// TIA Portal V16 export
// export: Created 2023-06-21T17:06:26.413978Z, ExportSetting WithDefaults, DisplayName Totally Integrated Automation Portal, DisplayVersion V16 Update 4, DisplayName TIA Portal Version Control Interface, DisplayVersion V16 Update 2, DisplayName TIA Portal Openness, DisplayVersion V16 Update 4, DisplayName SINAMICS Startdrive Advanced, DisplayVersion V16, DisplayName SINAMICS Startdrive G130, G150, S120, S150, SINAMICS MV, S210, DisplayVersion V16, DisplayName SINAMICS Startdrive G110M, G120, G120C, G120D, G120P, DisplayVersion V16, DisplayName STEP 7 Professional, DisplayVersion V16 Update 4, DisplayName STEP 7 Safety, DisplayVersion V16, DisplayName Soft Starter ES, DisplayVersion V16, DisplayName WinCC Advanced, DisplayVersion V16 Update 4
FUNCTION_BLOCK "MB_Comm_Setup"   // FB1, LAD
{ S7_Optimized_Access := 'FALSE' }
VERSION : 0.1
// stored: AutoNumber true, IsIECCheckEnabled false, SetENOAutomatically false, UDAEnableTagReadback false
   VAR DB_SPECIFIC
      Input_Registers_3000X_In { ExternalAccessible := 'False'; ExternalVisible := 'False'; ExternalWritable := 'False'} : Struct
         "3000X" { ExternalAccessible := 'False'; ExternalVisible := 'False'; ExternalWritable := 'False'} : Array[0..150] of Word;
      END_STRUCT;
   END_VAR
   VAR
      Input_Registers_In_AT AT Input_Registers_3000X_In : Struct
         "30001" : Array[0..15] of Bool;
         "30001_2" : Array[0..15] of Bool;   // Status of the Adaptor
         "30002" : Array[0..15] of Bool;   // Indoor Unit Connection Status
         "30003" : Array[0..15] of Bool;   // Empty
         "30004" : Array[0..15] of Bool;   // Empty
         "30005" : Array[0..15] of Bool;   // Empty
         "30006" : Array[0..15] of Bool;   // Indoor Unit Communication Status
         "31001" : Array[0..15] of Bool;   // Various
         "31002" : Array[0..15] of Bool;   // 1st word - Indoor unit cooling setpoint upper limit, 2 - word indoor unit cooling setpoint lower limit
         "31003" : Array[0..15] of Bool;   // 1st word - Indoor unit heating setpoint upper limit, 2 - word indoor unit heating setpoint lower limit
         "31004" : Array[0..15] of Bool;   // Various
         "31005" : Array[0..15] of Bool;   // 1st word - Indoor unit cooling setpoint upper limit, 2 - word indoor unit cooling setpoint lower limit
         "31006" : Array[0..15] of Bool;   // 1st word - Indoor unit heating setpoint upper limit, 2 - word indoor unit heating setpoint lower limit
         "31007" : Array[0..15] of Bool;   // Various
         "31008" : Array[0..15] of Bool;   // 1st word - Indoor unit cooling setpoint upper limit, 2 - word indoor unit cooling setpoint lower limit
         "31009" : Array[0..15] of Bool;   // 1st word - Indoor unit heating setpoint upper limit, 2 - word indoor unit heating setpoint lower limit
         "31010" : Array[0..15] of Bool;   // Various
         "31011" : Array[0..15] of Bool;   // 1st word - Indoor unit cooling setpoint upper limit, 2 - word indoor unit cooling setpoint lower limit
         "31012" : Array[0..15] of Bool;   // 1st word - Indoor unit heating setpoint upper limit, 2 - word indoor unit heating setpoint lower limit
         "31013" : Array[0..15] of Bool;   // Various
         "31014" : Array[0..15] of Bool;   // 1st word - Indoor unit cooling setpoint upper limit, 2 - word indoor unit cooling setpoint lower limit
         "31015" : Array[0..15] of Bool;   // 1st word - Indoor unit heating setpoint upper limit, 2 - word indoor unit heating setpoint lower limit
         "31016" : Array[0..15] of Bool;   // Various
         "31017" : Array[0..15] of Bool;   // 1st word - Indoor unit cooling setpoint upper limit, 2 - word indoor unit cooling setpoint lower limit
         "31018" : Array[0..15] of Bool;   // 1st word - Indoor unit heating setpoint upper limit, 2 - word indoor unit heating setpoint lower limit
         "31019" : Array[0..15] of Bool;   // Various
         "31020" : Array[0..15] of Bool;   // 1st word - Indoor unit cooling setpoint upper limit, 2 - word indoor unit cooling setpoint lower limit
         "31021" : Array[0..15] of Bool;   // 1st word - Indoor unit heating setpoint upper limit, 2 - word indoor unit heating setpoint lower limit
         "31022" : Array[0..15] of Bool;   // Various
         "31023" : Array[0..15] of Bool;   // 1st word - Indoor unit cooling setpoint upper limit, 2 - word indoor unit cooling setpoint lower limit
         "31024" : Array[0..15] of Bool;   // 1st word - Indoor unit heating setpoint upper limit, 2 - word indoor unit heating setpoint lower limit
         "31025" : Array[0..15] of Bool;   // Various
         "31026" : Array[0..15] of Bool;   // 1st word - Indoor unit cooling setpoint upper limit, 2 - word indoor unit cooling setpoint lower limit
         "31027" : Array[0..15] of Bool;   // 1st word - Indoor unit heating setpoint upper limit, 2 - word indoor unit heating setpoint lower limit
         "31028" : Array[0..15] of Bool;   // Various
         "31029" : Array[0..15] of Bool;   // 1st word - Indoor unit cooling setpoint upper limit, 2 - word indoor unit cooling setpoint lower limit
         "31030" : Array[0..15] of Bool;   // 1st word - Indoor unit heating setpoint upper limit, 2 - word indoor unit heating setpoint lower limit
         "31031" : Array[0..15] of Bool;   // Various
         "31032" : Array[0..15] of Bool;   // 1st word - Indoor unit cooling setpoint upper limit, 2 - word indoor unit cooling setpoint lower limit
         "31033" : Array[0..15] of Bool;   // 1st word - Indoor unit heating setpoint upper limit, 2 - word indoor unit heating setpoint lower limit
         "31034" : Array[0..15] of Bool;   // Various
         "31035" : Array[0..15] of Bool;   // 1st word - Indoor unit cooling setpoint upper limit, 2 - word indoor unit cooling setpoint lower limit
         "31036" : Array[0..15] of Bool;   // 1st word - Indoor unit heating setpoint upper limit, 2 - word indoor unit heating setpoint lower limit
         "31037" : Array[0..15] of Bool;   // Various
         "31038" : Array[0..15] of Bool;   // 1st word - Indoor unit cooling setpoint upper limit, 2 - word indoor unit cooling setpoint lower limit
         "31039" : Array[0..15] of Bool;   // 1st word - Indoor unit heating setpoint upper limit, 2 - word indoor unit heating setpoint lower limit
         "31040" : Array[0..15] of Bool;   // Various
         "31041" : Array[0..15] of Bool;   // 1st word - Indoor unit cooling setpoint upper limit, 2 - word indoor unit cooling setpoint lower limit
         "31042" : Array[0..15] of Bool;   // 1st word - Indoor unit heating setpoint upper limit, 2 - word indoor unit heating setpoint lower limit
         "31043" : Array[0..15] of Bool;   // Various
         "31044" : Array[0..15] of Bool;   // 1st word - Indoor unit cooling setpoint upper limit, 2 - word indoor unit cooling setpoint lower limit
         "31045" : Array[0..15] of Bool;   // 1st word - Indoor unit heating setpoint upper limit, 2 - word indoor unit heating setpoint lower limit
         "31046" : Array[0..15] of Bool;   // Various
         "31047" : Array[0..15] of Bool;   // 1st word - Indoor unit cooling setpoint upper limit, 2 - word indoor unit cooling setpoint lower limit
         "31048" : Array[0..15] of Bool;   // 1st word - Indoor unit heating setpoint upper limit, 2 - word indoor unit heating setpoint lower limit
         "32001" : Array[0..15] of Bool;   // Important stuff
         "32002" : Array[0..15] of Bool;   // Important stuff_2
         "32003" : Array[0..15] of Bool;   // Setpoint Temperature
         "32004" : Array[0..15] of Bool;   // Important Stuff_3
         "32005" : Array[0..15] of Bool;   // Room Temperature
         "32006" : Array[0..15] of Bool;   // Error
         "32007" : Array[0..15] of Bool;   // Important stuff
         "32008" : Array[0..15] of Bool;   // Important stuff_2
         "32009" : Array[0..15] of Bool;   // Setpoint Temperature
         "32010" : Array[0..15] of Bool;   // Important Stuff_3
         "32011" : Array[0..15] of Bool;   // Room Temperature
         "32012" : Array[0..15] of Bool;   // Error
         "32013" : Array[0..15] of Bool;   // Important stuff
         "32014" : Array[0..15] of Bool;   // Important stuff_2
         "32015" : Array[0..15] of Bool;   // Setpoint Temperature
         "32016" : Array[0..15] of Bool;   // Important Stuff_3
         "32017" : Array[0..15] of Bool;   // Room Temperature
         "32018" : Array[0..15] of Bool;   // Error
         "32019" : Array[0..15] of Bool;   // Important stuff
         "32020" : Array[0..15] of Bool;   // Important stuff_2
         "32021" : Array[0..15] of Bool;   // Setpoint Temperature
         "32022" : Array[0..15] of Bool;   // Important Stuff_3
         "32023" : Array[0..15] of Bool;   // Room Temperature
         "32024" : Array[0..15] of Bool;   // Error
         "32025" : Array[0..15] of Bool;   // Important stuff
         "32026" : Array[0..15] of Bool;   // Important stuff_2
         "32027" : Array[0..15] of Bool;   // Setpoint Temperature
         "32028" : Array[0..15] of Bool;   // Important Stuff_3
         "32029" : Array[0..15] of Bool;   // Room Temperature
         "32030" : Array[0..15] of Bool;   // Error
         "32031" : Array[0..15] of Bool;   // Important stuff
         "32032" : Array[0..15] of Bool;   // Important stuff_2
         "32033" : Array[0..15] of Bool;   // Setpoint Temperature
         "32034" : Array[0..15] of Bool;   // Important Stuff_3
         "32035" : Array[0..15] of Bool;   // Room Temperature
         "32036" : Array[0..15] of Bool;   // Error
         "32037" : Array[0..15] of Bool;   // Important stuff
         "32038" : Array[0..15] of Bool;   // Important stuff_2
         "32039" : Array[0..15] of Bool;   // Setpoint Temperature
         "32040" : Array[0..15] of Bool;   // Important Stuff_3
         "32041" : Array[0..15] of Bool;   // Room Temperature
         "32042" : Array[0..15] of Bool;   // Error
         "32043" : Array[0..15] of Bool;   // Important stuff
         "32044" : Array[0..15] of Bool;   // Important stuff_2
         "32045" : Array[0..15] of Bool;   // Setpoint Temperature
         "32046" : Array[0..15] of Bool;   // Important Stuff_3
         "32047" : Array[0..15] of Bool;   // Room Temperature
         "32048" : Array[0..15] of Bool;   // Error
         "32049" : Array[0..15] of Bool;   // Important stuff
         "32050" : Array[0..15] of Bool;   // Important stuff_2
         "32051" : Array[0..15] of Bool;   // Setpoint Temperature
         "32052" : Array[0..15] of Bool;   // Important Stuff_3
         "32053" : Array[0..15] of Bool;   // Room Temperature
         "32054" : Array[0..15] of Bool;   // Error
         "32055" : Array[0..15] of Bool;   // Important stuff
         "32056" : Array[0..15] of Bool;   // Important stuff_2
         "32057" : Array[0..15] of Bool;   // Setpoint Temperature
         "32058" : Array[0..15] of Bool;   // Important Stuff_3
         "32059" : Array[0..15] of Bool;   // Room Temperature
         "32060" : Array[0..15] of Bool;   // Error
         "32061" : Array[0..15] of Bool;   // Important stuff
         "32062" : Array[0..15] of Bool;   // Important stuff_2
         "32063" : Array[0..15] of Bool;   // Setpoint Temperature
         "32064" : Array[0..15] of Bool;   // Important Stuff_3
         "32065" : Array[0..15] of Bool;   // Room Temperature
         "32066" : Array[0..15] of Bool;   // Error
         "32067" : Array[0..15] of Bool;   // Important stuff
         "32068" : Array[0..15] of Bool;   // Important stuff_2
         "32069" : Array[0..15] of Bool;   // Setpoint Temperature
         "32070" : Array[0..15] of Bool;   // Important Stuff_3
         "32071" : Array[0..15] of Bool;   // Room Temperature
         "32072" : Array[0..15] of Bool;   // Error
         "32073" : Array[0..15] of Bool;   // Important stuff
         "32074" : Array[0..15] of Bool;   // Important stuff_2
         "32075" : Array[0..15] of Bool;   // Setpoint Temperature
         "32076" : Array[0..15] of Bool;   // Important Stuff_3
         "32077" : Array[0..15] of Bool;   // Room Temperature
         "32078" : Array[0..15] of Bool;   // Error
         "32079" : Array[0..15] of Bool;   // Important stuff
         "32080" : Array[0..15] of Bool;   // Important stuff_2
         "32081" : Array[0..15] of Bool;   // Setpoint Temperature
         "32082" : Array[0..15] of Bool;   // Important Stuff_3
         "32083" : Array[0..15] of Bool;   // Room Temperature
         "32084" : Array[0..15] of Bool;   // Error
         "32085" : Array[0..15] of Bool;   // Important stuff
         "32086" : Array[0..15] of Bool;   // Important stuff_2
         "32087" : Array[0..15] of Bool;   // Setpoint Temperature
         "32088" : Array[0..15] of Bool;   // Important Stuff_3
         "32089" : Array[0..15] of Bool;   // Room Temperature
         "32090" : Array[0..15] of Bool;   // Error
         "32091" : Array[0..15] of Bool;   // Important stuff
         "32092" : Array[0..15] of Bool;   // Important stuff_2
         "32093" : Array[0..15] of Bool;   // Setpoint Temperature
         "32094" : Array[0..15] of Bool;   // Important Stuff_3
         "32095" : Array[0..15] of Bool;   // Room Temperature
         "32096" : Array[0..15] of Bool;   // Error
      END_STRUCT;
   END_VAR
   // // Input_Registers_3000X_In."3000X"[0] : 30001
   // // Input_Registers_In_AT."30004"[0] : Fan Mode Capability
   // // Input_Registers_In_AT."30004"[1] : Cooling Mode Capability
   // // Input_Registers_In_AT."30004"[2] : Heating Mode Capability
   // // Input_Registers_In_AT."30004"[3] : Auto Mode Capability
   // // Input_Registers_In_AT."30004"[4] : Dry Mode Capability
   // // Input_Registers_In_AT."30004"[8] : Fan Direction Level Capability
   // // Input_Registers_In_AT."30004"[9] : Fan Direction Level Capability
   // // Input_Registers_In_AT."30004"[10] : Fan Direction Level Capability
   // // Input_Registers_In_AT."30004"[11] : Fan Direction Capability
   // // Input_Registers_In_AT."30004"[12] : Fan Volume Level Capability
   // // Input_Registers_In_AT."30004"[13] : Fan Volume Level Capability
   // // Input_Registers_In_AT."30004"[14] : Fan Volume Level Capability
   // // Input_Registers_In_AT."30004"[15] : Fan Volume Capability
   // // Input_Registers_In_AT."30005"[0] : Fan Mode Capability
   // // Input_Registers_In_AT."30005"[1] : Cooling Mode Capability
   // // Input_Registers_In_AT."30005"[2] : Heating Mode Capability
   // // Input_Registers_In_AT."30005"[3] : Auto Mode Capability
   // // Input_Registers_In_AT."30005"[4] : Dry Mode Capability
   // // Input_Registers_In_AT."30005"[8] : Fan Direction Level Capability
   // // Input_Registers_In_AT."30005"[9] : Fan Direction Level Capability
   // // Input_Registers_In_AT."30005"[10] : Fan Direction Level Capability
   // // Input_Registers_In_AT."30005"[11] : Fan Direction Capability
   // // Input_Registers_In_AT."30005"[12] : Fan Volume Level Capability
   // // Input_Registers_In_AT."30005"[13] : Fan Volume Level Capability
   // // Input_Registers_In_AT."30005"[14] : Fan Volume Level Capability
   // // Input_Registers_In_AT."30005"[15] : Fan Volume Capability
   // // Input_Registers_In_AT."31001"[0] : Fan Mode Capability
   // // Input_Registers_In_AT."31001"[1] : Cooling Mode Capability
   // // Input_Registers_In_AT."31001"[2] : Heating Mode Capability
   // // Input_Registers_In_AT."31001"[3] : Auto Mode Capability
   // // Input_Registers_In_AT."31001"[4] : Dry Mode Capability
   // // Input_Registers_In_AT."31001"[8] : Fan Direction Level Capability
   // // Input_Registers_In_AT."31001"[9] : Fan Direction Level Capability
   // // Input_Registers_In_AT."31001"[10] : Fan Direction Level Capability
   // // Input_Registers_In_AT."31001"[11] : Fan Direction Capability
   // // Input_Registers_In_AT."31001"[12] : Fan Volume Level Capability
   // // Input_Registers_In_AT."31001"[13] : Fan Volume Level Capability
   // // Input_Registers_In_AT."31001"[14] : Fan Volume Level Capability
   // // Input_Registers_In_AT."31001"[15] : Fan Volume Capability
   // // Input_Registers_In_AT."31004"[0] : Fan Mode Capability
   // // Input_Registers_In_AT."31004"[1] : Cooling Mode Capability
   // // Input_Registers_In_AT."31004"[2] : Heating Mode Capability
   // // Input_Registers_In_AT."31004"[3] : Auto Mode Capability
   // // Input_Registers_In_AT."31004"[4] : Dry Mode Capability
   // // Input_Registers_In_AT."31004"[8] : Fan Direction Level Capability
   // // Input_Registers_In_AT."31004"[9] : Fan Direction Level Capability
   // // Input_Registers_In_AT."31004"[10] : Fan Direction Level Capability
   // // Input_Registers_In_AT."31004"[11] : Fan Direction Capability
   // // Input_Registers_In_AT."31004"[12] : Fan Volume Level Capability
   // // Input_Registers_In_AT."31004"[13] : Fan Volume Level Capability
   // // Input_Registers_In_AT."31004"[14] : Fan Volume Level Capability
   // // Input_Registers_In_AT."31004"[15] : Fan Volume Capability
   // // Input_Registers_In_AT."31007"[0] : Fan Mode Capability
   // // Input_Registers_In_AT."31007"[1] : Cooling Mode Capability
   // // Input_Registers_In_AT."31007"[2] : Heating Mode Capability
   // // Input_Registers_In_AT."31007"[3] : Auto Mode Capability
   // // Input_Registers_In_AT."31007"[4] : Dry Mode Capability
   // // Input_Registers_In_AT."31007"[8] : Fan Direction Level Capability
   // // Input_Registers_In_AT."31007"[9] : Fan Direction Level Capability
   // // Input_Registers_In_AT."31007"[10] : Fan Direction Level Capability
   // // Input_Registers_In_AT."31007"[11] : Fan Direction Capability
   // // Input_Registers_In_AT."31007"[12] : Fan Volume Level Capability
   // // Input_Registers_In_AT."31007"[13] : Fan Volume Level Capability
   // // Input_Registers_In_AT."31007"[14] : Fan Volume Level Capability
   // // Input_Registers_In_AT."31007"[15] : Fan Volume Capability
   // // Input_Registers_In_AT."31010"[0] : Fan Mode Capability
   // // Input_Registers_In_AT."31010"[1] : Cooling Mode Capability
   // // Input_Registers_In_AT."31010"[2] : Heating Mode Capability
   // // Input_Registers_In_AT."31010"[3] : Auto Mode Capability
   // // Input_Registers_In_AT."31010"[4] : Dry Mode Capability
   // // Input_Registers_In_AT."31010"[8] : Fan Direction Level Capability
   // // Input_Registers_In_AT."31010"[9] : Fan Direction Level Capability
   // // Input_Registers_In_AT."31010"[10] : Fan Direction Level Capability
   // // Input_Registers_In_AT."31010"[11] : Fan Direction Capability
   // // Input_Registers_In_AT."31010"[12] : Fan Volume Level Capability
   // // Input_Registers_In_AT."31010"[13] : Fan Volume Level Capability
   // // Input_Registers_In_AT."31010"[14] : Fan Volume Level Capability
   // // Input_Registers_In_AT."31010"[15] : Fan Volume Capability
   // // Input_Registers_In_AT."31013"[0] : Fan Mode Capability
   // // Input_Registers_In_AT."31013"[1] : Cooling Mode Capability
   // // Input_Registers_In_AT."31013"[2] : Heating Mode Capability
   // // Input_Registers_In_AT."31013"[3] : Auto Mode Capability
   // // Input_Registers_In_AT."31013"[4] : Dry Mode Capability
   // // Input_Registers_In_AT."31013"[8] : Fan Direction Level Capability
   // // Input_Registers_In_AT."31013"[9] : Fan Direction Level Capability
   // // Input_Registers_In_AT."31013"[10] : Fan Direction Level Capability
   // // Input_Registers_In_AT."31013"[11] : Fan Direction Capability
   // // Input_Registers_In_AT."31013"[12] : Fan Volume Level Capability
   // // Input_Registers_In_AT."31013"[13] : Fan Volume Level Capability
   // // Input_Registers_In_AT."31013"[14] : Fan Volume Level Capability
   // // Input_Registers_In_AT."31013"[15] : Fan Volume Capability
   // // Input_Registers_In_AT."31016"[0] : Fan Mode Capability
   // // Input_Registers_In_AT."31016"[1] : Cooling Mode Capability
   // // Input_Registers_In_AT."31016"[2] : Heating Mode Capability
   // // Input_Registers_In_AT."31016"[3] : Auto Mode Capability
   // // Input_Registers_In_AT."31016"[4] : Dry Mode Capability
   // // Input_Registers_In_AT."31016"[8] : Fan Direction Level Capability
   // // Input_Registers_In_AT."31016"[9] : Fan Direction Level Capability
   // // Input_Registers_In_AT."31016"[10] : Fan Direction Level Capability
   // // Input_Registers_In_AT."31016"[11] : Fan Direction Capability
   // // Input_Registers_In_AT."31016"[12] : Fan Volume Level Capability
   // // Input_Registers_In_AT."31016"[13] : Fan Volume Level Capability
   // // Input_Registers_In_AT."31016"[14] : Fan Volume Level Capability
   // // Input_Registers_In_AT."31016"[15] : Fan Volume Capability
   // // Input_Registers_In_AT."31019"[0] : Fan Mode Capability
   // // Input_Registers_In_AT."31019"[1] : Cooling Mode Capability
   // // Input_Registers_In_AT."31019"[2] : Heating Mode Capability
   // // Input_Registers_In_AT."31019"[3] : Auto Mode Capability
   // // Input_Registers_In_AT."31019"[4] : Dry Mode Capability
   // // Input_Registers_In_AT."31019"[8] : Fan Direction Level Capability
   // // Input_Registers_In_AT."31019"[9] : Fan Direction Level Capability
   // // Input_Registers_In_AT."31019"[10] : Fan Direction Level Capability
   // // Input_Registers_In_AT."31019"[11] : Fan Direction Capability
   // // Input_Registers_In_AT."31019"[12] : Fan Volume Level Capability
   // // Input_Registers_In_AT."31019"[13] : Fan Volume Level Capability
   // // Input_Registers_In_AT."31019"[14] : Fan Volume Level Capability
   // // Input_Registers_In_AT."31019"[15] : Fan Volume Capability
   // // Input_Registers_In_AT."31022"[0] : Fan Mode Capability
   // // Input_Registers_In_AT."31022"[1] : Cooling Mode Capability
   // // Input_Registers_In_AT."31022"[2] : Heating Mode Capability
   // // Input_Registers_In_AT."31022"[3] : Auto Mode Capability
   // // Input_Registers_In_AT."31022"[4] : Dry Mode Capability
   // // Input_Registers_In_AT."31022"[8] : Fan Direction Level Capability
   // // Input_Registers_In_AT."31022"[9] : Fan Direction Level Capability
   // // Input_Registers_In_AT."31022"[10] : Fan Direction Level Capability
   // // Input_Registers_In_AT."31022"[11] : Fan Direction Capability
   // // Input_Registers_In_AT."31022"[12] : Fan Volume Level Capability
   // // Input_Registers_In_AT."31022"[13] : Fan Volume Level Capability
   // // Input_Registers_In_AT."31022"[14] : Fan Volume Level Capability
   // // Input_Registers_In_AT."31022"[15] : Fan Volume Capability
   // // Input_Registers_In_AT."31025"[0] : Fan Mode Capability
   // // Input_Registers_In_AT."31025"[1] : Cooling Mode Capability
   // // Input_Registers_In_AT."31025"[2] : Heating Mode Capability
   // // Input_Registers_In_AT."31025"[3] : Auto Mode Capability
   // // Input_Registers_In_AT."31025"[4] : Dry Mode Capability
   // // Input_Registers_In_AT."31025"[8] : Fan Direction Level Capability
   // // Input_Registers_In_AT."31025"[9] : Fan Direction Level Capability
   // // Input_Registers_In_AT."31025"[10] : Fan Direction Level Capability
   // // Input_Registers_In_AT."31025"[11] : Fan Direction Capability
   // // Input_Registers_In_AT."31025"[12] : Fan Volume Level Capability
   // // Input_Registers_In_AT."31025"[13] : Fan Volume Level Capability
   // // Input_Registers_In_AT."31025"[14] : Fan Volume Level Capability
   // // Input_Registers_In_AT."31025"[15] : Fan Volume Capability
   // // Input_Registers_In_AT."31028"[0] : Fan Mode Capability
   // // Input_Registers_In_AT."31028"[1] : Cooling Mode Capability
   // // Input_Registers_In_AT."31028"[2] : Heating Mode Capability
   // // Input_Registers_In_AT."31028"[3] : Auto Mode Capability
   // // Input_Registers_In_AT."31028"[4] : Dry Mode Capability
   // // Input_Registers_In_AT."31028"[8] : Fan Direction Level Capability
   // // Input_Registers_In_AT."31028"[9] : Fan Direction Level Capability
   // // Input_Registers_In_AT."31028"[10] : Fan Direction Level Capability
   // // Input_Registers_In_AT."31028"[11] : Fan Direction Capability
   // // Input_Registers_In_AT."31028"[12] : Fan Volume Level Capability
   // // Input_Registers_In_AT."31028"[13] : Fan Volume Level Capability
   // // Input_Registers_In_AT."31028"[14] : Fan Volume Level Capability
   // // Input_Registers_In_AT."31028"[15] : Fan Volume Capability
   // // Input_Registers_In_AT."31031"[0] : Fan Mode Capability
   // // Input_Registers_In_AT."31031"[1] : Cooling Mode Capability
   // // Input_Registers_In_AT."31031"[2] : Heating Mode Capability
   // // Input_Registers_In_AT."31031"[3] : Auto Mode Capability
   // // Input_Registers_In_AT."31031"[4] : Dry Mode Capability
   // // Input_Registers_In_AT."31031"[8] : Fan Direction Level Capability
   // // Input_Registers_In_AT."31031"[9] : Fan Direction Level Capability
   // // Input_Registers_In_AT."31031"[10] : Fan Direction Level Capability
   // // Input_Registers_In_AT."31031"[11] : Fan Direction Capability
   // // Input_Registers_In_AT."31031"[12] : Fan Volume Level Capability
   // // Input_Registers_In_AT."31031"[13] : Fan Volume Level Capability
   // // Input_Registers_In_AT."31031"[14] : Fan Volume Level Capability
   // // Input_Registers_In_AT."31031"[15] : Fan Volume Capability
   // // Input_Registers_In_AT."31034"[0] : Fan Mode Capability
   // // Input_Registers_In_AT."31034"[1] : Cooling Mode Capability
   // // Input_Registers_In_AT."31034"[2] : Heating Mode Capability
   // // Input_Registers_In_AT."31034"[3] : Auto Mode Capability
   // // Input_Registers_In_AT."31034"[4] : Dry Mode Capability
   // // Input_Registers_In_AT."31034"[8] : Fan Direction Level Capability
   // // Input_Registers_In_AT."31034"[9] : Fan Direction Level Capability
   // // Input_Registers_In_AT."31034"[10] : Fan Direction Level Capability
   // // Input_Registers_In_AT."31034"[11] : Fan Direction Capability
   // // Input_Registers_In_AT."31034"[12] : Fan Volume Level Capability
   // // Input_Registers_In_AT."31034"[13] : Fan Volume Level Capability
   // // Input_Registers_In_AT."31034"[14] : Fan Volume Level Capability
   // // Input_Registers_In_AT."31034"[15] : Fan Volume Capability
   // // Input_Registers_In_AT."31037"[0] : Fan Mode Capability
   // // Input_Registers_In_AT."31037"[1] : Cooling Mode Capability
   // // Input_Registers_In_AT."31037"[2] : Heating Mode Capability
   // // Input_Registers_In_AT."31037"[3] : Auto Mode Capability
   // // Input_Registers_In_AT."31037"[4] : Dry Mode Capability
   // // Input_Registers_In_AT."31037"[8] : Fan Direction Level Capability
   // // Input_Registers_In_AT."31037"[9] : Fan Direction Level Capability
   // // Input_Registers_In_AT."31037"[10] : Fan Direction Level Capability
   // // Input_Registers_In_AT."31037"[11] : Fan Direction Capability
   // // Input_Registers_In_AT."31037"[12] : Fan Volume Level Capability
   // // Input_Registers_In_AT."31037"[13] : Fan Volume Level Capability
   // // Input_Registers_In_AT."31037"[14] : Fan Volume Level Capability
   // // Input_Registers_In_AT."31037"[15] : Fan Volume Capability
   // // Input_Registers_In_AT."31040"[0] : Fan Mode Capability
   // // Input_Registers_In_AT."31040"[1] : Cooling Mode Capability
   // // Input_Registers_In_AT."31040"[2] : Heating Mode Capability
   // // Input_Registers_In_AT."31040"[3] : Auto Mode Capability
   // // Input_Registers_In_AT."31040"[4] : Dry Mode Capability
   // // Input_Registers_In_AT."31040"[8] : Fan Direction Level Capability
   // // Input_Registers_In_AT."31040"[9] : Fan Direction Level Capability
   // // Input_Registers_In_AT."31040"[10] : Fan Direction Level Capability
   // // Input_Registers_In_AT."31040"[11] : Fan Direction Capability
   // // Input_Registers_In_AT."31040"[12] : Fan Volume Level Capability
   // // Input_Registers_In_AT."31040"[13] : Fan Volume Level Capability
   // // Input_Registers_In_AT."31040"[14] : Fan Volume Level Capability
   // // Input_Registers_In_AT."31040"[15] : Fan Volume Capability
   // // Input_Registers_In_AT."31043"[0] : Fan Mode Capability
   // // Input_Registers_In_AT."31043"[1] : Cooling Mode Capability
   // // Input_Registers_In_AT."31043"[2] : Heating Mode Capability
   // // Input_Registers_In_AT."31043"[3] : Auto Mode Capability
   // // Input_Registers_In_AT."31043"[4] : Dry Mode Capability
   // // Input_Registers_In_AT."31043"[8] : Fan Direction Level Capability
   // // Input_Registers_In_AT."31043"[9] : Fan Direction Level Capability
   // // Input_Registers_In_AT."31043"[10] : Fan Direction Level Capability
   // // Input_Registers_In_AT."31043"[11] : Fan Direction Capability
   // // Input_Registers_In_AT."31043"[12] : Fan Volume Level Capability
   // // Input_Registers_In_AT."31043"[13] : Fan Volume Level Capability
   // // Input_Registers_In_AT."31043"[14] : Fan Volume Level Capability
   // // Input_Registers_In_AT."31043"[15] : Fan Volume Capability
   // // Input_Registers_In_AT."31046"[0] : Fan Mode Capability
   // // Input_Registers_In_AT."31046"[1] : Cooling Mode Capability
   // // Input_Registers_In_AT."31046"[2] : Heating Mode Capability
   // // Input_Registers_In_AT."31046"[3] : Auto Mode Capability
   // // Input_Registers_In_AT."31046"[4] : Dry Mode Capability
   // // Input_Registers_In_AT."31046"[8] : Fan Direction Level Capability
   // // Input_Registers_In_AT."31046"[9] : Fan Direction Level Capability
   // // Input_Registers_In_AT."31046"[10] : Fan Direction Level Capability
   // // Input_Registers_In_AT."31046"[11] : Fan Direction Capability
   // // Input_Registers_In_AT."31046"[12] : Fan Volume Level Capability
   // // Input_Registers_In_AT."31046"[13] : Fan Volume Level Capability
   // // Input_Registers_In_AT."31046"[14] : Fan Volume Level Capability
   // // Input_Registers_In_AT."31046"[15] : Fan Volume Capability
   // // Input_Registers_In_AT."32001"[0] : OnOff Status
   // // Input_Registers_In_AT."32001"[2] : Forced off status
   // // Input_Registers_In_AT."32001"[8] : Fan direction
   // // Input_Registers_In_AT."32001"[9] : Fan direction
   // // Input_Registers_In_AT."32001"[10] : Fan direction
   // // Input_Registers_In_AT."32001"[12] : Fan volume
   // // Input_Registers_In_AT."32001"[13] : Fan volume
   // // Input_Registers_In_AT."32001"[14] : Fan volume
   // // Input_Registers_In_AT."32002"[0] : Operation mode
   // // Input_Registers_In_AT."32002"[1] : Operation mode
   // // Input_Registers_In_AT."32002"[2] : Operation mode
   // // Input_Registers_In_AT."32002"[3] : Operation mode
   // // Input_Registers_In_AT."32002"[4] : Filter sign status
   // // Input_Registers_In_AT."32002"[5] : Filter sign status
   // // Input_Registers_In_AT."32002"[6] : Filter sign status
   // // Input_Registers_In_AT."32002"[7] : Filter sign status
   // // Input_Registers_In_AT."32002"[8] : Operation status
   // // Input_Registers_In_AT."32002"[9] : Operation status
   // // Input_Registers_In_AT."32002"[10] : Operation status
   // // Input_Registers_In_AT."32002"[11] : Operation status
   // // Input_Registers_In_AT."32002"[14] : Cool/Heat Master
   // // Input_Registers_In_AT."32002"[15] : Cool/Heat Master
   // // Input_Registers_In_AT."32003"[15] : Signed Bit
   // // Input_Registers_In_AT."32004"[0] : Error code mapping value1
   // // Input_Registers_In_AT."32004"[1] : Error code mapping value1
   // // Input_Registers_In_AT."32004"[2] : Error code mapping value1
   // // Input_Registers_In_AT."32004"[3] : Error code mapping value1
   // // Input_Registers_In_AT."32004"[4] : Error code mapping value2
   // // Input_Registers_In_AT."32004"[5] : Error code mapping value2
   // // Input_Registers_In_AT."32004"[6] : Error code mapping value2
   // // Input_Registers_In_AT."32004"[7] : Error code mapping value2
   // // Input_Registers_In_AT."32004"[8] : Malfunction
   // // Input_Registers_In_AT."32004"[9] : Warning
   // // Input_Registers_In_AT."32004"[10] : Operation status
   // // Input_Registers_In_AT."32005"[15] : Signed Bit
   // // Input_Registers_In_AT."32006"[8] : Indoor unit temperature sensor error
   // // Input_Registers_In_AT."32006"[15] : Indoor unit temperature sensor data received
   // // Input_Registers_In_AT."32007"[0] : OnOff Status
   // // Input_Registers_In_AT."32007"[2] : Forced off status
   // // Input_Registers_In_AT."32007"[8] : Fan direction
   // // Input_Registers_In_AT."32007"[9] : Fan direction
   // // Input_Registers_In_AT."32007"[10] : Fan direction
   // // Input_Registers_In_AT."32007"[12] : Fan volume
   // // Input_Registers_In_AT."32007"[13] : Fan volume
   // // Input_Registers_In_AT."32007"[14] : Fan volume
   // // Input_Registers_In_AT."32008"[0] : Operation mode
   // // Input_Registers_In_AT."32008"[1] : Operation mode
   // // Input_Registers_In_AT."32008"[2] : Operation mode
   // // Input_Registers_In_AT."32008"[3] : Operation mode
   // // Input_Registers_In_AT."32008"[4] : Filter sign status
   // // Input_Registers_In_AT."32008"[5] : Filter sign status
   // // Input_Registers_In_AT."32008"[6] : Filter sign status
   // // Input_Registers_In_AT."32008"[7] : Filter sign status
   // // Input_Registers_In_AT."32008"[8] : Operation status
   // // Input_Registers_In_AT."32008"[9] : Operation status
   // // Input_Registers_In_AT."32008"[10] : Operation status
   // // Input_Registers_In_AT."32008"[11] : Operation status
   // // Input_Registers_In_AT."32008"[14] : Cool/Heat Master
   // // Input_Registers_In_AT."32008"[15] : Cool/Heat Master
   // // Input_Registers_In_AT."32009"[15] : Signed Bit
   // // Input_Registers_In_AT."32010"[0] : Error code mapping value1
   // // Input_Registers_In_AT."32010"[1] : Error code mapping value1
   // // Input_Registers_In_AT."32010"[2] : Error code mapping value1
   // // Input_Registers_In_AT."32010"[3] : Error code mapping value1
   // // Input_Registers_In_AT."32010"[4] : Error code mapping value2
   // // Input_Registers_In_AT."32010"[5] : Error code mapping value2
   // // Input_Registers_In_AT."32010"[6] : Error code mapping value2
   // // Input_Registers_In_AT."32010"[7] : Error code mapping value2
   // // Input_Registers_In_AT."32010"[8] : Malfunction
   // // Input_Registers_In_AT."32010"[9] : Warning
   // // Input_Registers_In_AT."32010"[10] : Operation status
   // // Input_Registers_In_AT."32011"[15] : Signed Bit
   // // Input_Registers_In_AT."32012"[8] : Indoor unit temperature sensor error
   // // Input_Registers_In_AT."32012"[15] : Indoor unit temperature sensor data received
   // // Input_Registers_In_AT."32013"[0] : OnOff Status
   // // Input_Registers_In_AT."32013"[2] : Forced off status
   // // Input_Registers_In_AT."32013"[8] : Fan direction
   // // Input_Registers_In_AT."32013"[9] : Fan direction
   // // Input_Registers_In_AT."32013"[10] : Fan direction
   // // Input_Registers_In_AT."32013"[12] : Fan volume
   // // Input_Registers_In_AT."32013"[13] : Fan volume
   // // Input_Registers_In_AT."32013"[14] : Fan volume
   // // Input_Registers_In_AT."32014"[0] : Operation mode
   // // Input_Registers_In_AT."32014"[1] : Operation mode
   // // Input_Registers_In_AT."32014"[2] : Operation mode
   // // Input_Registers_In_AT."32014"[3] : Operation mode
   // // Input_Registers_In_AT."32014"[4] : Filter sign status
   // // Input_Registers_In_AT."32014"[5] : Filter sign status
   // // Input_Registers_In_AT."32014"[6] : Filter sign status
   // // Input_Registers_In_AT."32014"[7] : Filter sign status
   // // Input_Registers_In_AT."32014"[8] : Operation status
   // // Input_Registers_In_AT."32014"[9] : Operation status
   // // Input_Registers_In_AT."32014"[10] : Operation status
   // // Input_Registers_In_AT."32014"[11] : Operation status
   // // Input_Registers_In_AT."32014"[14] : Cool/Heat Master
   // // Input_Registers_In_AT."32014"[15] : Cool/Heat Master
   // // Input_Registers_In_AT."32015"[15] : Signed Bit
   // // Input_Registers_In_AT."32016"[0] : Error code mapping value1
   // // Input_Registers_In_AT."32016"[1] : Error code mapping value1
   // // Input_Registers_In_AT."32016"[2] : Error code mapping value1
   // // Input_Registers_In_AT."32016"[3] : Error code mapping value1
   // // Input_Registers_In_AT."32016"[4] : Error code mapping value2
   // // Input_Registers_In_AT."32016"[5] : Error code mapping value2
   // // Input_Registers_In_AT."32016"[6] : Error code mapping value2
   // // Input_Registers_In_AT."32016"[7] : Error code mapping value2
   // // Input_Registers_In_AT."32016"[8] : Malfunction
   // // Input_Registers_In_AT."32016"[9] : Warning
   // // Input_Registers_In_AT."32016"[10] : Operation status
   // // Input_Registers_In_AT."32017"[15] : Signed Bit
   // // Input_Registers_In_AT."32018"[8] : Indoor unit temperature sensor error
   // // Input_Registers_In_AT."32018"[15] : Indoor unit temperature sensor data received
   // // Input_Registers_In_AT."32019"[0] : OnOff Status
   // // Input_Registers_In_AT."32019"[2] : Forced off status
   // // Input_Registers_In_AT."32019"[8] : Fan direction
   // // Input_Registers_In_AT."32019"[9] : Fan direction
   // // Input_Registers_In_AT."32019"[10] : Fan direction
   // // Input_Registers_In_AT."32019"[12] : Fan volume
   // // Input_Registers_In_AT."32019"[13] : Fan volume
   // // Input_Registers_In_AT."32019"[14] : Fan volume
   // // Input_Registers_In_AT."32020"[0] : Operation mode
   // // Input_Registers_In_AT."32020"[1] : Operation mode
   // // Input_Registers_In_AT."32020"[2] : Operation mode
   // // Input_Registers_In_AT."32020"[3] : Operation mode
   // // Input_Registers_In_AT."32020"[4] : Filter sign status
   // // Input_Registers_In_AT."32020"[5] : Filter sign status
   // // Input_Registers_In_AT."32020"[6] : Filter sign status
   // // Input_Registers_In_AT."32020"[7] : Filter sign status
   // // Input_Registers_In_AT."32020"[8] : Operation status
   // // Input_Registers_In_AT."32020"[9] : Operation status
   // // Input_Registers_In_AT."32020"[10] : Operation status
   // // Input_Registers_In_AT."32020"[11] : Operation status
   // // Input_Registers_In_AT."32020"[14] : Cool/Heat Master
   // // Input_Registers_In_AT."32020"[15] : Cool/Heat Master
   // // Input_Registers_In_AT."32021"[15] : Signed Bit
   // // Input_Registers_In_AT."32022"[0] : Error code mapping value1
   // // Input_Registers_In_AT."32022"[1] : Error code mapping value1
   // // Input_Registers_In_AT."32022"[2] : Error code mapping value1
   // // Input_Registers_In_AT."32022"[3] : Error code mapping value1
   // // Input_Registers_In_AT."32022"[4] : Error code mapping value2
   // // Input_Registers_In_AT."32022"[5] : Error code mapping value2
   // // Input_Registers_In_AT."32022"[6] : Error code mapping value2
   // // Input_Registers_In_AT."32022"[7] : Error code mapping value2
   // // Input_Registers_In_AT."32022"[8] : Malfunction
   // // Input_Registers_In_AT."32022"[9] : Warning
   // // Input_Registers_In_AT."32022"[10] : Operation status
   // // Input_Registers_In_AT."32023"[15] : Signed Bit
   // // Input_Registers_In_AT."32024"[8] : Indoor unit temperature sensor error
   // // Input_Registers_In_AT."32024"[15] : Indoor unit temperature sensor data received
   // // Input_Registers_In_AT."32025"[0] : OnOff Status
   // // Input_Registers_In_AT."32025"[2] : Forced off status
   // // Input_Registers_In_AT."32025"[8] : Fan direction
   // // Input_Registers_In_AT."32025"[9] : Fan direction
   // // Input_Registers_In_AT."32025"[10] : Fan direction
   // // Input_Registers_In_AT."32025"[12] : Fan volume
   // // Input_Registers_In_AT."32025"[13] : Fan volume
   // // Input_Registers_In_AT."32025"[14] : Fan volume
   // // Input_Registers_In_AT."32026"[0] : Operation mode
   // // Input_Registers_In_AT."32026"[1] : Operation mode
   // // Input_Registers_In_AT."32026"[2] : Operation mode
   // // Input_Registers_In_AT."32026"[3] : Operation mode
   // // Input_Registers_In_AT."32026"[4] : Filter sign status
   // // Input_Registers_In_AT."32026"[5] : Filter sign status
   // // Input_Registers_In_AT."32026"[6] : Filter sign status
   // // Input_Registers_In_AT."32026"[7] : Filter sign status
   // // Input_Registers_In_AT."32026"[8] : Operation status
   // // Input_Registers_In_AT."32026"[9] : Operation status
   // // Input_Registers_In_AT."32026"[10] : Operation status
   // // Input_Registers_In_AT."32026"[11] : Operation status
   // // Input_Registers_In_AT."32026"[14] : Cool/Heat Master
   // // Input_Registers_In_AT."32026"[15] : Cool/Heat Master
   // // Input_Registers_In_AT."32027"[15] : Signed Bit
   // // Input_Registers_In_AT."32028"[0] : Error code mapping value1
   // // Input_Registers_In_AT."32028"[1] : Error code mapping value1
   // // Input_Registers_In_AT."32028"[2] : Error code mapping value1
   // // Input_Registers_In_AT."32028"[3] : Error code mapping value1
   // // Input_Registers_In_AT."32028"[4] : Error code mapping value2
   // // Input_Registers_In_AT."32028"[5] : Error code mapping value2
   // // Input_Registers_In_AT."32028"[6] : Error code mapping value2
   // // Input_Registers_In_AT."32028"[7] : Error code mapping value2
   // // Input_Registers_In_AT."32028"[8] : Malfunction
   // // Input_Registers_In_AT."32028"[9] : Warning
   // // Input_Registers_In_AT."32028"[10] : Operation status
   // // Input_Registers_In_AT."32029"[15] : Signed Bit
   // // Input_Registers_In_AT."32030"[8] : Indoor unit temperature sensor error
   // // Input_Registers_In_AT."32030"[15] : Indoor unit temperature sensor data received
   // // Input_Registers_In_AT."32031"[0] : OnOff Status
   // // Input_Registers_In_AT."32031"[2] : Forced off status
   // // Input_Registers_In_AT."32031"[8] : Fan direction
   // // Input_Registers_In_AT."32031"[9] : Fan direction
   // // Input_Registers_In_AT."32031"[10] : Fan direction
   // // Input_Registers_In_AT."32031"[12] : Fan volume
   // // Input_Registers_In_AT."32031"[13] : Fan volume
   // // Input_Registers_In_AT."32031"[14] : Fan volume
   // // Input_Registers_In_AT."32032"[0] : Operation mode
   // // Input_Registers_In_AT."32032"[1] : Operation mode
   // // Input_Registers_In_AT."32032"[2] : Operation mode
   // // Input_Registers_In_AT."32032"[3] : Operation mode
   // // Input_Registers_In_AT."32032"[4] : Filter sign status
   // // Input_Registers_In_AT."32032"[5] : Filter sign status
   // // Input_Registers_In_AT."32032"[6] : Filter sign status
   // // Input_Registers_In_AT."32032"[7] : Filter sign status
   // // Input_Registers_In_AT."32032"[8] : Operation status
   // // Input_Registers_In_AT."32032"[9] : Operation status
   // // Input_Registers_In_AT."32032"[10] : Operation status
   // // Input_Registers_In_AT."32032"[11] : Operation status
   // // Input_Registers_In_AT."32032"[14] : Cool/Heat Master
   // // Input_Registers_In_AT."32032"[15] : Cool/Heat Master
   // // Input_Registers_In_AT."32033"[15] : Signed Bit
   // // Input_Registers_In_AT."32034"[0] : Error code mapping value1
   // // Input_Registers_In_AT."32034"[1] : Error code mapping value1
   // // Input_Registers_In_AT."32034"[2] : Error code mapping value1
   // // Input_Registers_In_AT."32034"[3] : Error code mapping value1
   // // Input_Registers_In_AT."32034"[4] : Error code mapping value2
   // // Input_Registers_In_AT."32034"[5] : Error code mapping value2
   // // Input_Registers_In_AT."32034"[6] : Error code mapping value2
   // // Input_Registers_In_AT."32034"[7] : Error code mapping value2
   // // Input_Registers_In_AT."32034"[8] : Malfunction
   // // Input_Registers_In_AT."32034"[9] : Warning
   // // Input_Registers_In_AT."32034"[10] : Operation status
   // // Input_Registers_In_AT."32035"[15] : Signed Bit
   // // Input_Registers_In_AT."32036"[8] : Indoor unit temperature sensor error
   // // Input_Registers_In_AT."32036"[15] : Indoor unit temperature sensor data received
   // // Input_Registers_In_AT."32037"[0] : OnOff Status
   // // Input_Registers_In_AT."32037"[2] : Forced off status
   // // Input_Registers_In_AT."32037"[8] : Fan direction
   // // Input_Registers_In_AT."32037"[9] : Fan direction
   // // Input_Registers_In_AT."32037"[10] : Fan direction
   // // Input_Registers_In_AT."32037"[12] : Fan volume
   // // Input_Registers_In_AT."32037"[13] : Fan volume
   // // Input_Registers_In_AT."32037"[14] : Fan volume
   // // Input_Registers_In_AT."32038"[0] : Operation mode
   // // Input_Registers_In_AT."32038"[1] : Operation mode
   // // Input_Registers_In_AT."32038"[2] : Operation mode
   // // Input_Registers_In_AT."32038"[3] : Operation mode
   // // Input_Registers_In_AT."32038"[4] : Filter sign status
   // // Input_Registers_In_AT."32038"[5] : Filter sign status
   // // Input_Registers_In_AT."32038"[6] : Filter sign status
   // // Input_Registers_In_AT."32038"[7] : Filter sign status
   // // Input_Registers_In_AT."32038"[8] : Operation status
   // // Input_Registers_In_AT."32038"[9] : Operation status
   // // Input_Registers_In_AT."32038"[10] : Operation status
   // // Input_Registers_In_AT."32038"[11] : Operation status
   // // Input_Registers_In_AT."32038"[14] : Cool/Heat Master
   // // Input_Registers_In_AT."32038"[15] : Cool/Heat Master
   // // Input_Registers_In_AT."32039"[15] : Signed Bit
   // // Input_Registers_In_AT."32040"[0] : Error code mapping value1
   // // Input_Registers_In_AT."32040"[1] : Error code mapping value1
   // // Input_Registers_In_AT."32040"[2] : Error code mapping value1
   // // Input_Registers_In_AT."32040"[3] : Error code mapping value1
   // // Input_Registers_In_AT."32040"[4] : Error code mapping value2
   // // Input_Registers_In_AT."32040"[5] : Error code mapping value2
   // // Input_Registers_In_AT."32040"[6] : Error code mapping value2
   // // Input_Registers_In_AT."32040"[7] : Error code mapping value2
   // // Input_Registers_In_AT."32040"[8] : Malfunction
   // // Input_Registers_In_AT."32040"[9] : Warning
   // // Input_Registers_In_AT."32040"[10] : Operation status
   // // Input_Registers_In_AT."32041"[15] : Signed Bit
   // // Input_Registers_In_AT."32042"[8] : Indoor unit temperature sensor error
   // // Input_Registers_In_AT."32042"[15] : Indoor unit temperature sensor data received
   // // Input_Registers_In_AT."32043"[0] : OnOff Status
   // // Input_Registers_In_AT."32043"[2] : Forced off status
   // // Input_Registers_In_AT."32043"[8] : Fan direction
   // // Input_Registers_In_AT."32043"[9] : Fan direction
   // // Input_Registers_In_AT."32043"[10] : Fan direction
   // // Input_Registers_In_AT."32043"[12] : Fan volume
   // // Input_Registers_In_AT."32043"[13] : Fan volume
   // // Input_Registers_In_AT."32043"[14] : Fan volume
   // // Input_Registers_In_AT."32044"[0] : Operation mode
   // // Input_Registers_In_AT."32044"[1] : Operation mode
   // // Input_Registers_In_AT."32044"[2] : Operation mode
   // // Input_Registers_In_AT."32044"[3] : Operation mode
   // // Input_Registers_In_AT."32044"[4] : Filter sign status
   // // Input_Registers_In_AT."32044"[5] : Filter sign status
   // // Input_Registers_In_AT."32044"[6] : Filter sign status
   // // Input_Registers_In_AT."32044"[7] : Filter sign status
   // // Input_Registers_In_AT."32044"[8] : Operation status
   // // Input_Registers_In_AT."32044"[9] : Operation status
   // // Input_Registers_In_AT."32044"[10] : Operation status
   // // Input_Registers_In_AT."32044"[11] : Operation status
   // // Input_Registers_In_AT."32044"[14] : Cool/Heat Master
   // // Input_Registers_In_AT."32044"[15] : Cool/Heat Master
   // // Input_Registers_In_AT."32045"[15] : Signed Bit
   // // Input_Registers_In_AT."32046"[0] : Error code mapping value1
   // // Input_Registers_In_AT."32046"[1] : Error code mapping value1
   // // Input_Registers_In_AT."32046"[2] : Error code mapping value1
   // // Input_Registers_In_AT."32046"[3] : Error code mapping value1
   // // Input_Registers_In_AT."32046"[4] : Error code mapping value2
   // // Input_Registers_In_AT."32046"[5] : Error code mapping value2
   // // Input_Registers_In_AT."32046"[6] : Error code mapping value2
   // // Input_Registers_In_AT."32046"[7] : Error code mapping value2
   // // Input_Registers_In_AT."32046"[8] : Malfunction
   // // Input_Registers_In_AT."32046"[9] : Warning
   // // Input_Registers_In_AT."32046"[10] : Operation status
   // // Input_Registers_In_AT."32047"[15] : Signed Bit
   // // Input_Registers_In_AT."32048"[8] : Indoor unit temperature sensor error
   // // Input_Registers_In_AT."32048"[15] : Indoor unit temperature sensor data received
   // // Input_Registers_In_AT."32049"[0] : OnOff Status
   // // Input_Registers_In_AT."32049"[2] : Forced off status
   // // Input_Registers_In_AT."32049"[8] : Fan direction
   // // Input_Registers_In_AT."32049"[9] : Fan direction
   // // Input_Registers_In_AT."32049"[10] : Fan direction
   // // Input_Registers_In_AT."32049"[12] : Fan volume
   // // Input_Registers_In_AT."32049"[13] : Fan volume
   // // Input_Registers_In_AT."32049"[14] : Fan volume
   // // Input_Registers_In_AT."32050"[0] : Operation mode
   // // Input_Registers_In_AT."32050"[1] : Operation mode
   // // Input_Registers_In_AT."32050"[2] : Operation mode
   // // Input_Registers_In_AT."32050"[3] : Operation mode
   // // Input_Registers_In_AT."32050"[4] : Filter sign status
   // // Input_Registers_In_AT."32050"[5] : Filter sign status
   // // Input_Registers_In_AT."32050"[6] : Filter sign status
   // // Input_Registers_In_AT."32050"[7] : Filter sign status
   // // Input_Registers_In_AT."32050"[8] : Operation status
   // // Input_Registers_In_AT."32050"[9] : Operation status
   // // Input_Registers_In_AT."32050"[10] : Operation status
   // // Input_Registers_In_AT."32050"[11] : Operation status
   // // Input_Registers_In_AT."32050"[14] : Cool/Heat Master
   // // Input_Registers_In_AT."32050"[15] : Cool/Heat Master
   // // Input_Registers_In_AT."32051"[15] : Signed Bit
   // // Input_Registers_In_AT."32052"[0] : Error code mapping value1
   // // Input_Registers_In_AT."32052"[1] : Error code mapping value1
   // // Input_Registers_In_AT."32052"[2] : Error code mapping value1
   // // Input_Registers_In_AT."32052"[3] : Error code mapping value1
   // // Input_Registers_In_AT."32052"[4] : Error code mapping value2
   // // Input_Registers_In_AT."32052"[5] : Error code mapping value2
   // // Input_Registers_In_AT."32052"[6] : Error code mapping value2
   // // Input_Registers_In_AT."32052"[7] : Error code mapping value2
   // // Input_Registers_In_AT."32052"[8] : Malfunction
   // // Input_Registers_In_AT."32052"[9] : Warning
   // // Input_Registers_In_AT."32052"[10] : Operation status
   // // Input_Registers_In_AT."32053"[15] : Signed Bit
   // // Input_Registers_In_AT."32054"[8] : Indoor unit temperature sensor error
   // // Input_Registers_In_AT."32054"[15] : Indoor unit temperature sensor data received
   // // Input_Registers_In_AT."32055"[0] : OnOff Status
   // // Input_Registers_In_AT."32055"[2] : Forced off status
   // // Input_Registers_In_AT."32055"[8] : Fan direction
   // // Input_Registers_In_AT."32055"[9] : Fan direction
   // // Input_Registers_In_AT."32055"[10] : Fan direction
   // // Input_Registers_In_AT."32055"[12] : Fan volume
   // // Input_Registers_In_AT."32055"[13] : Fan volume
   // // Input_Registers_In_AT."32055"[14] : Fan volume
   // // Input_Registers_In_AT."32056"[0] : Operation mode
   // // Input_Registers_In_AT."32056"[1] : Operation mode
   // // Input_Registers_In_AT."32056"[2] : Operation mode
   // // Input_Registers_In_AT."32056"[3] : Operation mode
   // // Input_Registers_In_AT."32056"[4] : Filter sign status
   // // Input_Registers_In_AT."32056"[5] : Filter sign status
   // // Input_Registers_In_AT."32056"[6] : Filter sign status
   // // Input_Registers_In_AT."32056"[7] : Filter sign status
   // // Input_Registers_In_AT."32056"[8] : Operation status
   // // Input_Registers_In_AT."32056"[9] : Operation status
   // // Input_Registers_In_AT."32056"[10] : Operation status
   // // Input_Registers_In_AT."32056"[11] : Operation status
   // // Input_Registers_In_AT."32056"[14] : Cool/Heat Master
   // // Input_Registers_In_AT."32056"[15] : Cool/Heat Master
   // // Input_Registers_In_AT."32057"[15] : Signed Bit
   // // Input_Registers_In_AT."32058"[0] : Error code mapping value1
   // // Input_Registers_In_AT."32058"[1] : Error code mapping value1
   // // Input_Registers_In_AT."32058"[2] : Error code mapping value1
   // // Input_Registers_In_AT."32058"[3] : Error code mapping value1
   // // Input_Registers_In_AT."32058"[4] : Error code mapping value2
   // // Input_Registers_In_AT."32058"[5] : Error code mapping value2
   // // Input_Registers_In_AT."32058"[6] : Error code mapping value2
   // // Input_Registers_In_AT."32058"[7] : Error code mapping value2
   // // Input_Registers_In_AT."32058"[8] : Malfunction
   // // Input_Registers_In_AT."32058"[9] : Warning
   // // Input_Registers_In_AT."32058"[10] : Operation status
   // // Input_Registers_In_AT."32059"[15] : Signed Bit
   // // Input_Registers_In_AT."32060"[8] : Indoor unit temperature sensor error
   // // Input_Registers_In_AT."32060"[15] : Indoor unit temperature sensor data received
   // // Input_Registers_In_AT."32061"[0] : OnOff Status
   // // Input_Registers_In_AT."32061"[2] : Forced off status
   // // Input_Registers_In_AT."32061"[8] : Fan direction
   // // Input_Registers_In_AT."32061"[9] : Fan direction
   // // Input_Registers_In_AT."32061"[10] : Fan direction
   // // Input_Registers_In_AT."32061"[12] : Fan volume
   // // Input_Registers_In_AT."32061"[13] : Fan volume
   // // Input_Registers_In_AT."32061"[14] : Fan volume
   // // Input_Registers_In_AT."32062"[0] : Operation mode
   // // Input_Registers_In_AT."32062"[1] : Operation mode
   // // Input_Registers_In_AT."32062"[2] : Operation mode
   // // Input_Registers_In_AT."32062"[3] : Operation mode
   // // Input_Registers_In_AT."32062"[4] : Filter sign status
   // // Input_Registers_In_AT."32062"[5] : Filter sign status
   // // Input_Registers_In_AT."32062"[6] : Filter sign status
   // // Input_Registers_In_AT."32062"[7] : Filter sign status
   // // Input_Registers_In_AT."32062"[8] : Operation status
   // // Input_Registers_In_AT."32062"[9] : Operation status
   // // Input_Registers_In_AT."32062"[10] : Operation status
   // // Input_Registers_In_AT."32062"[11] : Operation status
   // // Input_Registers_In_AT."32062"[14] : Cool/Heat Master
   // // Input_Registers_In_AT."32062"[15] : Cool/Heat Master
   // // Input_Registers_In_AT."32063"[15] : Signed Bit
   // // Input_Registers_In_AT."32064"[0] : Error code mapping value1
   // // Input_Registers_In_AT."32064"[1] : Error code mapping value1
   // // Input_Registers_In_AT."32064"[2] : Error code mapping value1
   // // Input_Registers_In_AT."32064"[3] : Error code mapping value1
   // // Input_Registers_In_AT."32064"[4] : Error code mapping value2
   // // Input_Registers_In_AT."32064"[5] : Error code mapping value2
   // // Input_Registers_In_AT."32064"[6] : Error code mapping value2
   // // Input_Registers_In_AT."32064"[7] : Error code mapping value2
   // // Input_Registers_In_AT."32064"[8] : Malfunction
   // // Input_Registers_In_AT."32064"[9] : Warning
   // // Input_Registers_In_AT."32064"[10] : Operation status
   // // Input_Registers_In_AT."32065"[15] : Signed Bit
   // // Input_Registers_In_AT."32066"[8] : Indoor unit temperature sensor error
   // // Input_Registers_In_AT."32066"[15] : Indoor unit temperature sensor data received
   // // Input_Registers_In_AT."32067"[0] : OnOff Status
   // // Input_Registers_In_AT."32067"[2] : Forced off status
   // // Input_Registers_In_AT."32067"[8] : Fan direction
   // // Input_Registers_In_AT."32067"[9] : Fan direction
   // // Input_Registers_In_AT."32067"[10] : Fan direction
   // // Input_Registers_In_AT."32067"[12] : Fan volume
   // // Input_Registers_In_AT."32067"[13] : Fan volume
   // // Input_Registers_In_AT."32067"[14] : Fan volume
   // // Input_Registers_In_AT."32068"[0] : Operation mode
   // // Input_Registers_In_AT."32068"[1] : Operation mode
   // // Input_Registers_In_AT."32068"[2] : Operation mode
   // // Input_Registers_In_AT."32068"[3] : Operation mode
   // // Input_Registers_In_AT."32068"[4] : Filter sign status
   // // Input_Registers_In_AT."32068"[5] : Filter sign status
   // // Input_Registers_In_AT."32068"[6] : Filter sign status
   // // Input_Registers_In_AT."32068"[7] : Filter sign status
   // // Input_Registers_In_AT."32068"[8] : Operation status
   // // Input_Registers_In_AT."32068"[9] : Operation status
   // // Input_Registers_In_AT."32068"[10] : Operation status
   // // Input_Registers_In_AT."32068"[11] : Operation status
   // // Input_Registers_In_AT."32068"[14] : Cool/Heat Master
   // // Input_Registers_In_AT."32068"[15] : Cool/Heat Master
   // // Input_Registers_In_AT."32069"[15] : Signed Bit
   // // Input_Registers_In_AT."32070"[0] : Error code mapping value1
   // // Input_Registers_In_AT."32070"[1] : Error code mapping value1
   // // Input_Registers_In_AT."32070"[2] : Error code mapping value1
   // // Input_Registers_In_AT."32070"[3] : Error code mapping value1
   // // Input_Registers_In_AT."32070"[4] : Error code mapping value2
   // // Input_Registers_In_AT."32070"[5] : Error code mapping value2
   // // Input_Registers_In_AT."32070"[6] : Error code mapping value2
   // // Input_Registers_In_AT."32070"[7] : Error code mapping value2
   // // Input_Registers_In_AT."32070"[8] : Malfunction
   // // Input_Registers_In_AT."32070"[9] : Warning
   // // Input_Registers_In_AT."32070"[10] : Operation status
   // // Input_Registers_In_AT."32071"[15] : Signed Bit
   // // Input_Registers_In_AT."32072"[8] : Indoor unit temperature sensor error
   // // Input_Registers_In_AT."32072"[15] : Indoor unit temperature sensor data received
   // // Input_Registers_In_AT."32073"[0] : OnOff Status
   // // Input_Registers_In_AT."32073"[2] : Forced off status
   // // Input_Registers_In_AT."32073"[8] : Fan direction
   // // Input_Registers_In_AT."32073"[9] : Fan direction
   // // Input_Registers_In_AT."32073"[10] : Fan direction
   // // Input_Registers_In_AT."32073"[12] : Fan volume
   // // Input_Registers_In_AT."32073"[13] : Fan volume
   // // Input_Registers_In_AT."32073"[14] : Fan volume
   // // Input_Registers_In_AT."32074"[0] : Operation mode
   // // Input_Registers_In_AT."32074"[1] : Operation mode
   // // Input_Registers_In_AT."32074"[2] : Operation mode
   // // Input_Registers_In_AT."32074"[3] : Operation mode
   // // Input_Registers_In_AT."32074"[4] : Filter sign status
   // // Input_Registers_In_AT."32074"[5] : Filter sign status
   // // Input_Registers_In_AT."32074"[6] : Filter sign status
   // // Input_Registers_In_AT."32074"[7] : Filter sign status
   // // Input_Registers_In_AT."32074"[8] : Operation status
   // // Input_Registers_In_AT."32074"[9] : Operation status
   // // Input_Registers_In_AT."32074"[10] : Operation status
   // // Input_Registers_In_AT."32074"[11] : Operation status
   // // Input_Registers_In_AT."32074"[14] : Cool/Heat Master
   // // Input_Registers_In_AT."32074"[15] : Cool/Heat Master
   // // Input_Registers_In_AT."32075"[15] : Signed Bit
   // // Input_Registers_In_AT."32076"[0] : Error code mapping value1
   // // Input_Registers_In_AT."32076"[1] : Error code mapping value1
   // // Input_Registers_In_AT."32076"[2] : Error code mapping value1
   // // Input_Registers_In_AT."32076"[3] : Error code mapping value1
   // // Input_Registers_In_AT."32076"[4] : Error code mapping value2
   // // Input_Registers_In_AT."32076"[5] : Error code mapping value2
   // // Input_Registers_In_AT."32076"[6] : Error code mapping value2
   // // Input_Registers_In_AT."32076"[7] : Error code mapping value2
   // // Input_Registers_In_AT."32076"[8] : Malfunction
   // // Input_Registers_In_AT."32076"[9] : Warning
   // // Input_Registers_In_AT."32076"[10] : Operation status
   // // Input_Registers_In_AT."32077"[15] : Signed Bit
   // // Input_Registers_In_AT."32078"[8] : Indoor unit temperature sensor error
   // // Input_Registers_In_AT."32078"[15] : Indoor unit temperature sensor data received
   // // Input_Registers_In_AT."32079"[0] : OnOff Status
   // // Input_Registers_In_AT."32079"[2] : Forced off status
   // // Input_Registers_In_AT."32079"[8] : Fan direction
   // // Input_Registers_In_AT."32079"[9] : Fan direction
   // // Input_Registers_In_AT."32079"[10] : Fan direction
   // // Input_Registers_In_AT."32079"[12] : Fan volume
   // // Input_Registers_In_AT."32079"[13] : Fan volume
   // // Input_Registers_In_AT."32079"[14] : Fan volume
   // // Input_Registers_In_AT."32080"[0] : Operation mode
   // // Input_Registers_In_AT."32080"[1] : Operation mode
   // // Input_Registers_In_AT."32080"[2] : Operation mode
   // // Input_Registers_In_AT."32080"[3] : Operation mode
   // // Input_Registers_In_AT."32080"[4] : Filter sign status
   // // Input_Registers_In_AT."32080"[5] : Filter sign status
   // // Input_Registers_In_AT."32080"[6] : Filter sign status
   // // Input_Registers_In_AT."32080"[7] : Filter sign status
   // // Input_Registers_In_AT."32080"[8] : Operation status
   // // Input_Registers_In_AT."32080"[9] : Operation status
   // // Input_Registers_In_AT."32080"[10] : Operation status
   // // Input_Registers_In_AT."32080"[11] : Operation status
   // // Input_Registers_In_AT."32080"[14] : Cool/Heat Master
   // // Input_Registers_In_AT."32080"[15] : Cool/Heat Master
   // // Input_Registers_In_AT."32081"[15] : Signed Bit
   // // Input_Registers_In_AT."32082"[0] : Error code mapping value1
   // // Input_Registers_In_AT."32082"[1] : Error code mapping value1
   // // Input_Registers_In_AT."32082"[2] : Error code mapping value1
   // // Input_Registers_In_AT."32082"[3] : Error code mapping value1
   // // Input_Registers_In_AT."32082"[4] : Error code mapping value2
   // // Input_Registers_In_AT."32082"[5] : Error code mapping value2
   // // Input_Registers_In_AT."32082"[6] : Error code mapping value2
   // // Input_Registers_In_AT."32082"[7] : Error code mapping value2
   // // Input_Registers_In_AT."32082"[8] : Malfunction
   // // Input_Registers_In_AT."32082"[9] : Warning
   // // Input_Registers_In_AT."32082"[10] : Operation status
   // // Input_Registers_In_AT."32083"[15] : Signed Bit
   // // Input_Registers_In_AT."32084"[8] : Indoor unit temperature sensor error
   // // Input_Registers_In_AT."32084"[15] : Indoor unit temperature sensor data received
   // // Input_Registers_In_AT."32085"[0] : OnOff Status
   // // Input_Registers_In_AT."32085"[2] : Forced off status
   // // Input_Registers_In_AT."32085"[8] : Fan direction
   // // Input_Registers_In_AT."32085"[9] : Fan direction
   // // Input_Registers_In_AT."32085"[10] : Fan direction
   // // Input_Registers_In_AT."32085"[12] : Fan volume
   // // Input_Registers_In_AT."32085"[13] : Fan volume
   // // Input_Registers_In_AT."32085"[14] : Fan volume
   // // Input_Registers_In_AT."32086"[0] : Operation mode
   // // Input_Registers_In_AT."32086"[1] : Operation mode
   // // Input_Registers_In_AT."32086"[2] : Operation mode
   // // Input_Registers_In_AT."32086"[3] : Operation mode
   // // Input_Registers_In_AT."32086"[4] : Filter sign status
   // // Input_Registers_In_AT."32086"[5] : Filter sign status
   // // Input_Registers_In_AT."32086"[6] : Filter sign status
   // // Input_Registers_In_AT."32086"[7] : Filter sign status
   // // Input_Registers_In_AT."32086"[8] : Operation status
   // // Input_Registers_In_AT."32086"[9] : Operation status
   // // Input_Registers_In_AT."32086"[10] : Operation status
   // // Input_Registers_In_AT."32086"[11] : Operation status
   // // Input_Registers_In_AT."32086"[14] : Cool/Heat Master
   // // Input_Registers_In_AT."32086"[15] : Cool/Heat Master
   // // Input_Registers_In_AT."32087"[15] : Signed Bit
   // // Input_Registers_In_AT."32088"[0] : Error code mapping value1
   // // Input_Registers_In_AT."32088"[1] : Error code mapping value1
   // // Input_Registers_In_AT."32088"[2] : Error code mapping value1
   // // Input_Registers_In_AT."32088"[3] : Error code mapping value1
   // // Input_Registers_In_AT."32088"[4] : Error code mapping value2
   // // Input_Registers_In_AT."32088"[5] : Error code mapping value2
   // // Input_Registers_In_AT."32088"[6] : Error code mapping value2
   // // Input_Registers_In_AT."32088"[7] : Error code mapping value2
   // // Input_Registers_In_AT."32088"[8] : Malfunction
   // // Input_Registers_In_AT."32088"[9] : Warning
   // // Input_Registers_In_AT."32088"[10] : Operation status
   // // Input_Registers_In_AT."32089"[15] : Signed Bit
   // // Input_Registers_In_AT."32090"[8] : Indoor unit temperature sensor error
   // // Input_Registers_In_AT."32090"[15] : Indoor unit temperature sensor data received
   // // Input_Registers_In_AT."32091"[0] : OnOff Status
   // // Input_Registers_In_AT."32091"[2] : Forced off status
   // // Input_Registers_In_AT."32091"[8] : Fan direction
   // // Input_Registers_In_AT."32091"[9] : Fan direction
   // // Input_Registers_In_AT."32091"[10] : Fan direction
   // // Input_Registers_In_AT."32091"[12] : Fan volume
   // // Input_Registers_In_AT."32091"[13] : Fan volume
   // // Input_Registers_In_AT."32091"[14] : Fan volume
   // // Input_Registers_In_AT."32092"[0] : Operation mode
   // // Input_Registers_In_AT."32092"[1] : Operation mode
   // // Input_Registers_In_AT."32092"[2] : Operation mode
   // // Input_Registers_In_AT."32092"[3] : Operation mode
   // // Input_Registers_In_AT."32092"[4] : Filter sign status
   // // Input_Registers_In_AT."32092"[5] : Filter sign status
   // // Input_Registers_In_AT."32092"[6] : Filter sign status
   // // Input_Registers_In_AT."32092"[7] : Filter sign status
   // // Input_Registers_In_AT."32092"[8] : Operation status
   // // Input_Registers_In_AT."32092"[9] : Operation status
   // // Input_Registers_In_AT."32092"[10] : Operation status
   // // Input_Registers_In_AT."32092"[11] : Operation status
   // // Input_Registers_In_AT."32092"[14] : Cool/Heat Master
   // // Input_Registers_In_AT."32092"[15] : Cool/Heat Master
   // // Input_Registers_In_AT."32093"[15] : Signed Bit
   // // Input_Registers_In_AT."32094"[0] : Error code mapping value1
   // // Input_Registers_In_AT."32094"[1] : Error code mapping value1
   // // Input_Registers_In_AT."32094"[2] : Error code mapping value1
   // // Input_Registers_In_AT."32094"[3] : Error code mapping value1
   // // Input_Registers_In_AT."32094"[4] : Error code mapping value2
   // // Input_Registers_In_AT."32094"[5] : Error code mapping value2
   // // Input_Registers_In_AT."32094"[6] : Error code mapping value2
   // // Input_Registers_In_AT."32094"[7] : Error code mapping value2
   // // Input_Registers_In_AT."32094"[8] : Malfunction
   // // Input_Registers_In_AT."32094"[9] : Warning
   // // Input_Registers_In_AT."32094"[10] : Operation status
   // // Input_Registers_In_AT."32095"[15] : Signed Bit
   // // Input_Registers_In_AT."32096"[8] : Indoor unit temperature sensor error
   // // Input_Registers_In_AT."32096"[15] : Indoor unit temperature sensor data received
BEGIN

REGION Network 2: Enable supply voltage diagnostic
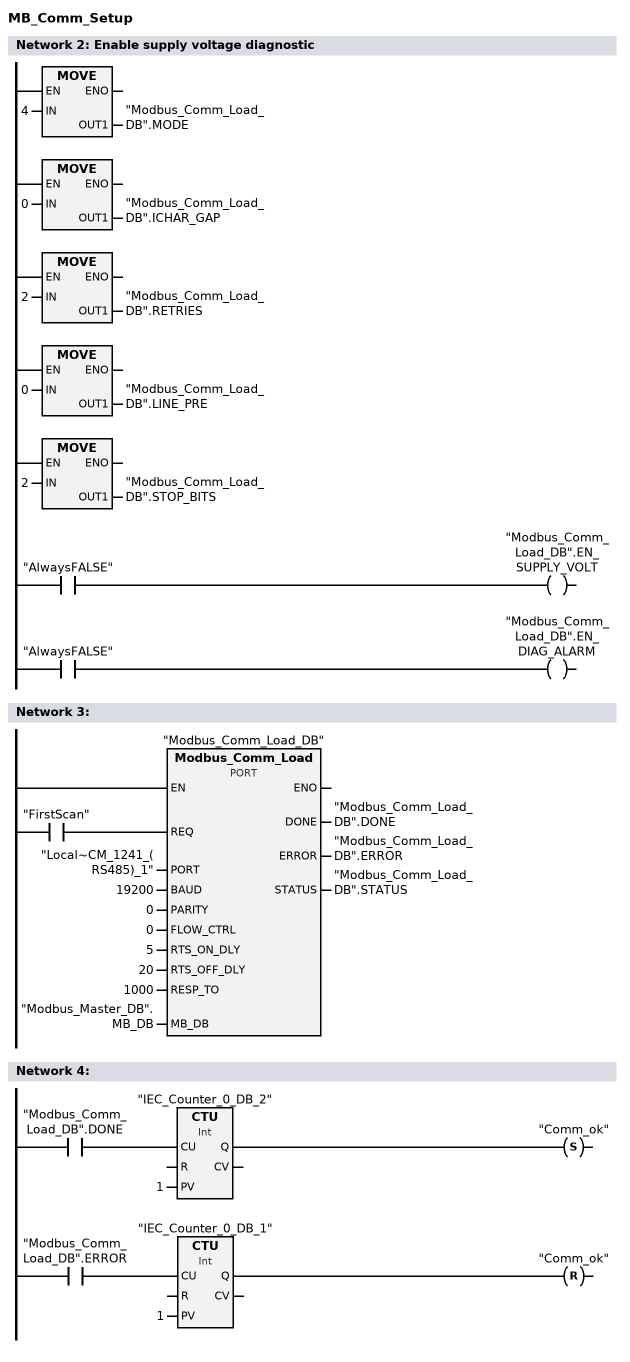
   RUNG wire#powerrail
      Move(in := 4, out1 => "Modbus_Comm_Load_DB".MODE)
   END_RUNG
   RUNG wire#powerrail
      Move(in := 0, out1 => "Modbus_Comm_Load_DB".ICHAR_GAP)
   END_RUNG
   RUNG wire#powerrail
      Move(in := 2, out1 => "Modbus_Comm_Load_DB".RETRIES)
   END_RUNG
   RUNG wire#powerrail
      Move(in := 0, out1 => "Modbus_Comm_Load_DB".LINE_PRE)
   END_RUNG
   RUNG wire#powerrail
      Move(in := 2, out1 => "Modbus_Comm_Load_DB".STOP_BITS)
   END_RUNG
   RUNG wire#powerrail
      Contact( "AlwaysFALSE" )
      Coil( "Modbus_Comm_Load_DB".EN_SUPPLY_VOLT )
   END_RUNG
   RUNG wire#powerrail
      Contact( "AlwaysFALSE" )
      Coil( "Modbus_Comm_Load_DB".EN_DIAG_ALARM )
   END_RUNG
   // the same network as SCL:
   "Modbus_Comm_Load_DB".MODE := 4;
   "Modbus_Comm_Load_DB".ICHAR_GAP := 0;
   "Modbus_Comm_Load_DB".RETRIES := 2;
   "Modbus_Comm_Load_DB".LINE_PRE := 0;
   "Modbus_Comm_Load_DB".STOP_BITS := 2;
   "Modbus_Comm_Load_DB".EN_SUPPLY_VOLT := "AlwaysFALSE";
   "Modbus_Comm_Load_DB".EN_DIAG_ALARM := "AlwaysFALSE";
END_REGION

REGION Network 3
   RUNG wire#powerrail
      { S7_Templates := "[card := 0, port_type := PORT, word_type := UInt, dint_type := UDInt, mbbase_type := P2P_MB_BASE]" } "Modbus_Comm_Load_DB".Modbus_Comm_Load(REQ := wire#w1, PORT := "Local~CM_1241_(RS485)_1", BAUD := 19200, PARITY := 0, FLOW_CTRL := 0, RTS_ON_DLY := 5, RTS_OFF_DLY := 20, RESP_TO := 1000, MB_DB := "Modbus_Master_DB".MB_DB, DONE => "Modbus_Comm_Load_DB".DONE, ERROR => "Modbus_Comm_Load_DB".ERROR, STATUS => "Modbus_Comm_Load_DB".STATUS)
   END_RUNG
   RUNG wire#powerrail
      Contact( "FirstScan" )
   END_RUNG wire#w1
   // the same network as SCL:
   "Modbus_Comm_Load_DB"(REQ := "FirstScan",   // Modbus_Comm_Load
                         PORT := "Local~CM_1241_(RS485)_1",
                         BAUD := 19200,
                         PARITY := 0,
                         FLOW_CTRL := 0,
                         RTS_ON_DLY := 5,
                         RTS_OFF_DLY := 20,
                         RESP_TO := 1000,
                         MB_DB := "Modbus_Master_DB".MB_DB,
                         DONE => "Modbus_Comm_Load_DB".DONE,
                         ERROR => "Modbus_Comm_Load_DB".ERROR,
                         STATUS => "Modbus_Comm_Load_DB".STATUS);
END_REGION

REGION Network 4
   RUNG wire#powerrail
      Contact( "Modbus_Comm_Load_DB".DONE )
      { S7_Templates := "value_type := Int" } "IEC_Counter_0_DB_2".CTU(r :=, pv := 1, cv =>)
      S_Coil( "Comm_ok" )
   END_RUNG
   RUNG wire#powerrail
      Contact( "Modbus_Comm_Load_DB".ERROR )
      { S7_Templates := "value_type := Int" } "IEC_Counter_0_DB_1".CTU(r :=, pv := 1, cv =>)
      R_Coil( "Comm_ok" )
   END_RUNG
   // the same network as SCL:
   "IEC_Counter_0_DB_2".CTU(CU := "Modbus_Comm_Load_DB".DONE, PV := 1);
   IF "IEC_Counter_0_DB_2".Q THEN "Comm_ok" := TRUE; END_IF;
   "IEC_Counter_0_DB_1".CTU(CU := "Modbus_Comm_Load_DB".ERROR, PV := 1);
   IF "IEC_Counter_0_DB_1".Q THEN "Comm_ok" := FALSE; END_IF;
END_REGION
END_FUNCTION_BLOCK
